PROGRAM Master1_IO_Map
VAR
	BYTE_AS_BIT_0: BYTE_AS_BIT;
	BYTE_AS_BIT_1: BYTE_AS_BIT;
	BYTE_AS_BIT_2: BYTE_AS_BIT;
	BYTE_AS_BIT_3: BYTE_AS_BIT;
	BYTE_AS_BIT_4: BYTE_AS_BIT;
	BYTE_AS_BIT_5: BYTE_AS_BIT;
	BYTE_AS_BIT_6: BYTE_AS_BIT;
	BYTE_AS_BIT_7: BYTE_AS_BIT;
	BYTE_AS_BIT_8: BYTE_AS_BIT;
	BYTE_AS_BIT_9: BYTE_AS_BIT;
	
	BIT_AS_BYTE_0: BIT_AS_BYTE;
	BIT_AS_BYTE_1: BIT_AS_BYTE;
	BIT_AS_BYTE_2: BIT_AS_BYTE;
	BIT_AS_BYTE_3: BIT_AS_BYTE;
	BIT_AS_BYTE_4: BIT_AS_BYTE;
	BIT_AS_BYTE_5: BIT_AS_BYTE;
	BIT_AS_BYTE_6: BIT_AS_BYTE;
	BIT_AS_BYTE_7: BIT_AS_BYTE;
	BIT_AS_BYTE_8: BIT_AS_BYTE;
	BIT_AS_BYTE_9: BIT_AS_BYTE;
	BIT_AS_BYTE_10: BIT_AS_BYTE;
	BIT_AS_BYTE_11: BIT_AS_BYTE;	
	
	OP10_MAS1_PORT1_BYTE1_DI_MODULE_1 AT %I* : BYTE;
	OP10_MAS1_PORT1_BYTE2_DI_MODULE_1 AT %I* : BYTE;
	OP10_MAS1_PORT2_BYTE1_DI_MODULE_2 AT %I* : BYTE;
	OP10_MAS1_PORT2_BYTE2_DI_MODULE_2 AT %I* : BYTE;
	OP10_MAS1_PORT3_BYTE1_DI_MODULE_3 AT %I* : BYTE;
	OP10_MAS1_PORT3_BYTE2_DI_MODULE_3 AT %I* : BYTE;
	OP10_MAS1_PORT4_BYTE1_DI_MODULE_4 AT %I* : BYTE;
	OP10_MAS1_PORT4_BYTE2_DI_MODULE_4 AT %I* : BYTE;
	OP10_MAS1_PORT5_BYTE1_DI_MODULE_5 AT %I* : BYTE;
	OP10_MAS1_PORT5_BYTE2_DI_MODULE_5 AT %I* : BYTE;
	
	OP10_MAS1_PORT6_BYTE1_DO_MODULE_1 AT %Q* : BYTE;
	OP10_MAS1_PORT6_BYTE2_DO_MODULE_1 AT %Q* : BYTE;
    OP10_MAS1_PORT6_BYTE3_DO_MODULE_1 AT %Q* : BYTE;
	OP10_MAS1_PORT6_BYTE4_DO_MODULE_1 AT %Q* : BYTE;
	
	OP10_MAS1_PORT7_BYTE1_DO_MODULE_2 AT %Q* : BYTE;
	OP10_MAS1_PORT7_BYTE2_DO_MODULE_2 AT %Q* : BYTE;
	OP10_MAS1_PORT7_BYTE3_DO_MODULE_2 AT %Q* : BYTE;
	OP10_MAS1_PORT7_BYTE4_DO_MODULE_2 AT %Q* : BYTE;
	
	OP10_MAS1_PORT8_BYTE1_DO_MODULE_3 AT %Q* : BYTE;
	OP10_MAS1_PORT8_BYTE2_DO_MODULE_3 AT %Q* : BYTE;
    OP10_MAS1_PORT8_BYTE3_DO_MODULE_3 AT %Q* : BYTE;
	OP10_MAS1_PORT8_BYTE4_DO_MODULE_3 AT %Q* : BYTE;
	
END_VAR

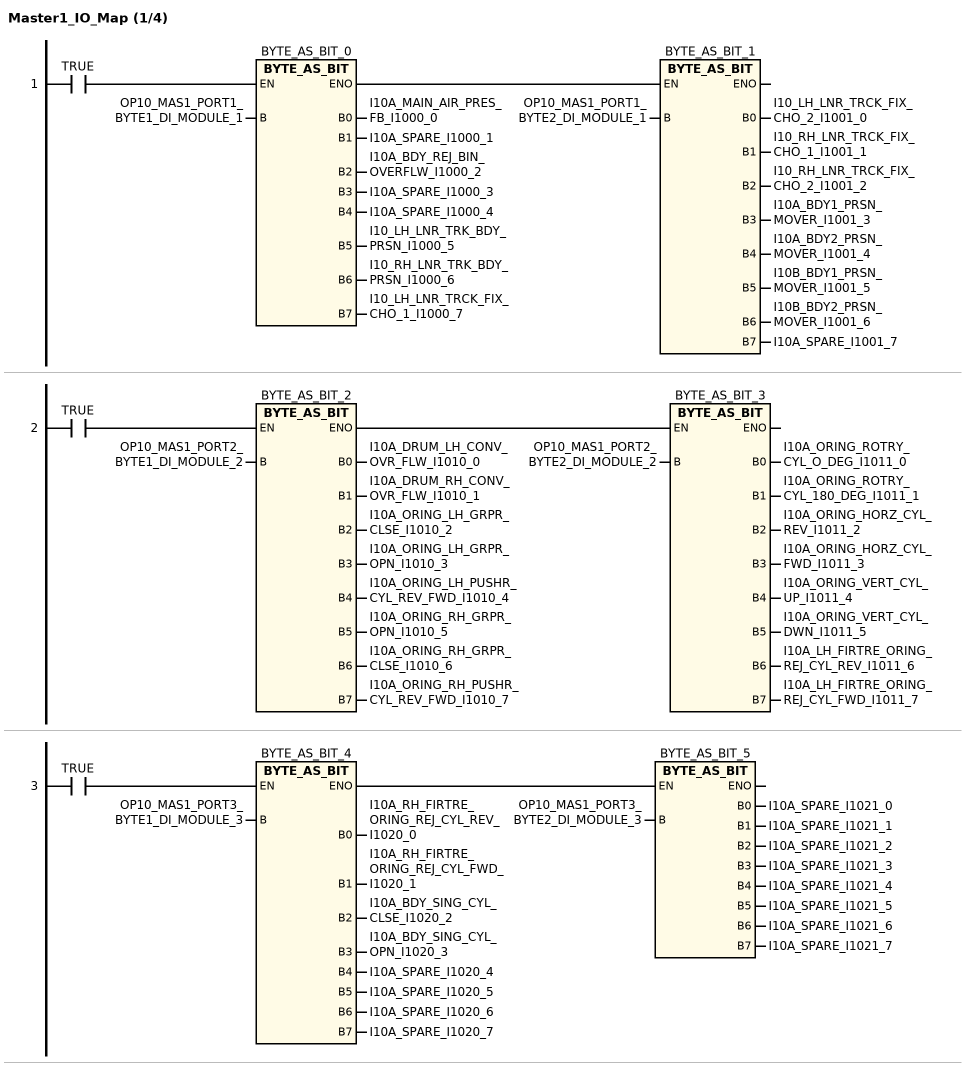
// NETWORK 1
BYTE_AS_BIT_0(
    B := OP10_MAS1_PORT1_BYTE1_DI_MODULE_1,
    B0 => I10A_MAIN_AIR_PRES_FB_I1000_0,
    B1 => I10A_SPARE_I1000_1,
    B2 => I10A_BDY_REJ_BIN_OVERFLW_I1000_2,
    B3 => I10A_SPARE_I1000_3,
    B4 => I10A_SPARE_I1000_4,
    B5 => I10_LH_LNR_TRK_BDY_PRSN_I1000_5,
    B6 => I10_RH_LNR_TRK_BDY_PRSN_I1000_6,
    B7 => I10_LH_LNR_TRCK_FIX_CHO_1_I1000_7); // BYTE_AS_BIT
BYTE_AS_BIT_1(
    B := OP10_MAS1_PORT1_BYTE2_DI_MODULE_1,
    B0 => I10_LH_LNR_TRCK_FIX_CHO_2_I1001_0,
    B1 => I10_RH_LNR_TRCK_FIX_CHO_1_I1001_1,
    B2 => I10_RH_LNR_TRCK_FIX_CHO_2_I1001_2,
    B3 => I10A_BDY1_PRSN_MOVER_I1001_3,
    B4 => I10A_BDY2_PRSN_MOVER_I1001_4,
    B5 => I10B_BDY1_PRSN_MOVER_I1001_5,
    B6 => I10B_BDY2_PRSN_MOVER_I1001_6,
    B7 => I10A_SPARE_I1001_7); // BYTE_AS_BIT

// NETWORK 2
BYTE_AS_BIT_2(
    B := OP10_MAS1_PORT2_BYTE1_DI_MODULE_2,
    B0 => I10A_DRUM_LH_CONV_OVR_FLW_I1010_0,
    B1 => I10A_DRUM_RH_CONV_OVR_FLW_I1010_1,
    B2 => I10A_ORING_LH_GRPR_CLSE_I1010_2,
    B3 => I10A_ORING_LH_GRPR_OPN_I1010_3,
    B4 => I10A_ORING_LH_PUSHR_CYL_REV_FWD_I1010_4,
    B5 => I10A_ORING_RH_GRPR_OPN_I1010_5,
    B6 => I10A_ORING_RH_GRPR_CLSE_I1010_6,
    B7 => I10A_ORING_RH_PUSHR_CYL_REV_FWD_I1010_7); // BYTE_AS_BIT
BYTE_AS_BIT_3(
    B := OP10_MAS1_PORT2_BYTE2_DI_MODULE_2,
    B0 => I10A_ORING_ROTRY_CYL_O_DEG_I1011_0,
    B1 => I10A_ORING_ROTRY_CYL_180_DEG_I1011_1,
    B2 => I10A_ORING_HORZ_CYL_REV_I1011_2,
    B3 => I10A_ORING_HORZ_CYL_FWD_I1011_3,
    B4 => I10A_ORING_VERT_CYL_UP_I1011_4,
    B5 => I10A_ORING_VERT_CYL_DWN_I1011_5,
    B6 => I10A_LH_FIRTRE_ORING_REJ_CYL_REV_I1011_6,
    B7 => I10A_LH_FIRTRE_ORING_REJ_CYL_FWD_I1011_7); // BYTE_AS_BIT

// NETWORK 3
BYTE_AS_BIT_4(
    B := OP10_MAS1_PORT3_BYTE1_DI_MODULE_3,
    B0 => I10A_RH_FIRTRE_ORING_REJ_CYL_REV_I1020_0,
    B1 => I10A_RH_FIRTRE_ORING_REJ_CYL_FWD_I1020_1,
    B2 => I10A_BDY_SING_CYL_CLSE_I1020_2,
    B3 => I10A_BDY_SING_CYL_OPN_I1020_3,
    B4 => I10A_SPARE_I1020_4,
    B5 => I10A_SPARE_I1020_5,
    B6 => I10A_SPARE_I1020_6,
    B7 => I10A_SPARE_I1020_7); // BYTE_AS_BIT
BYTE_AS_BIT_5(
    B := OP10_MAS1_PORT3_BYTE2_DI_MODULE_3,
    B0 => I10A_SPARE_I1021_0,
    B1 => I10A_SPARE_I1021_1,
    B2 => I10A_SPARE_I1021_2,
    B3 => I10A_SPARE_I1021_3,
    B4 => I10A_SPARE_I1021_4,
    B5 => I10A_SPARE_I1021_5,
    B6 => I10A_SPARE_I1021_6,
    B7 => I10A_SPARE_I1021_7); // BYTE_AS_BIT

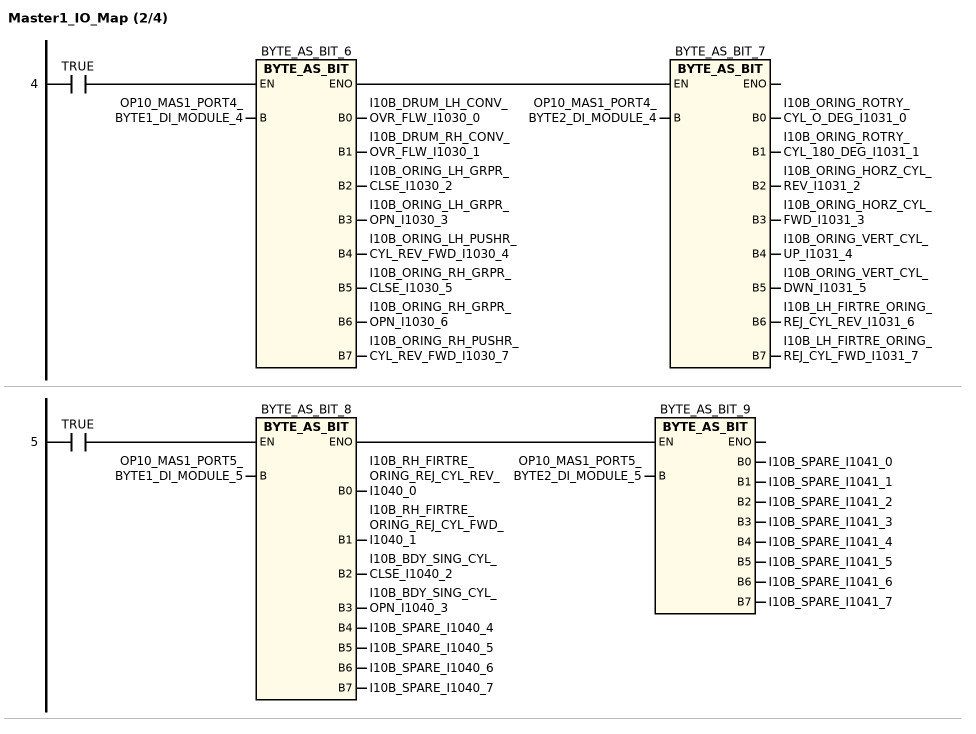
// NETWORK 4
BYTE_AS_BIT_6(
    B := OP10_MAS1_PORT4_BYTE1_DI_MODULE_4,
    B0 => I10B_DRUM_LH_CONV_OVR_FLW_I1030_0,
    B1 => I10B_DRUM_RH_CONV_OVR_FLW_I1030_1,
    B2 => I10B_ORING_LH_GRPR_CLSE_I1030_2,
    B3 => I10B_ORING_LH_GRPR_OPN_I1030_3,
    B4 => I10B_ORING_LH_PUSHR_CYL_REV_FWD_I1030_4,
    B5 => I10B_ORING_RH_GRPR_CLSE_I1030_5,
    B6 => I10B_ORING_RH_GRPR_OPN_I1030_6,
    B7 => I10B_ORING_RH_PUSHR_CYL_REV_FWD_I1030_7); // BYTE_AS_BIT
BYTE_AS_BIT_7(
    B := OP10_MAS1_PORT4_BYTE2_DI_MODULE_4,
    B0 => I10B_ORING_ROTRY_CYL_O_DEG_I1031_0,
    B1 => I10B_ORING_ROTRY_CYL_180_DEG_I1031_1,
    B2 => I10B_ORING_HORZ_CYL_REV_I1031_2,
    B3 => I10B_ORING_HORZ_CYL_FWD_I1031_3,
    B4 => I10B_ORING_VERT_CYL_UP_I1031_4,
    B5 => I10B_ORING_VERT_CYL_DWN_I1031_5,
    B6 => I10B_LH_FIRTRE_ORING_REJ_CYL_REV_I1031_6,
    B7 => I10B_LH_FIRTRE_ORING_REJ_CYL_FWD_I1031_7); // BYTE_AS_BIT

// NETWORK 5
BYTE_AS_BIT_8(
    B := OP10_MAS1_PORT5_BYTE1_DI_MODULE_5,
    B0 => I10B_RH_FIRTRE_ORING_REJ_CYL_REV_I1040_0,
    B1 => I10B_RH_FIRTRE_ORING_REJ_CYL_FWD_I1040_1,
    B2 => I10B_BDY_SING_CYL_CLSE_I1040_2,
    B3 => I10B_BDY_SING_CYL_OPN_I1040_3,
    B4 => I10B_SPARE_I1040_4,
    B5 => I10B_SPARE_I1040_5,
    B6 => I10B_SPARE_I1040_6,
    B7 => I10B_SPARE_I1040_7); // BYTE_AS_BIT
BYTE_AS_BIT_9(
    B := OP10_MAS1_PORT5_BYTE2_DI_MODULE_5,
    B0 => I10B_SPARE_I1041_0,
    B1 => I10B_SPARE_I1041_1,
    B2 => I10B_SPARE_I1041_2,
    B3 => I10B_SPARE_I1041_3,
    B4 => I10B_SPARE_I1041_4,
    B5 => I10B_SPARE_I1041_5,
    B6 => I10B_SPARE_I1041_6,
    B7 => I10B_SPARE_I1041_7); // BYTE_AS_BIT

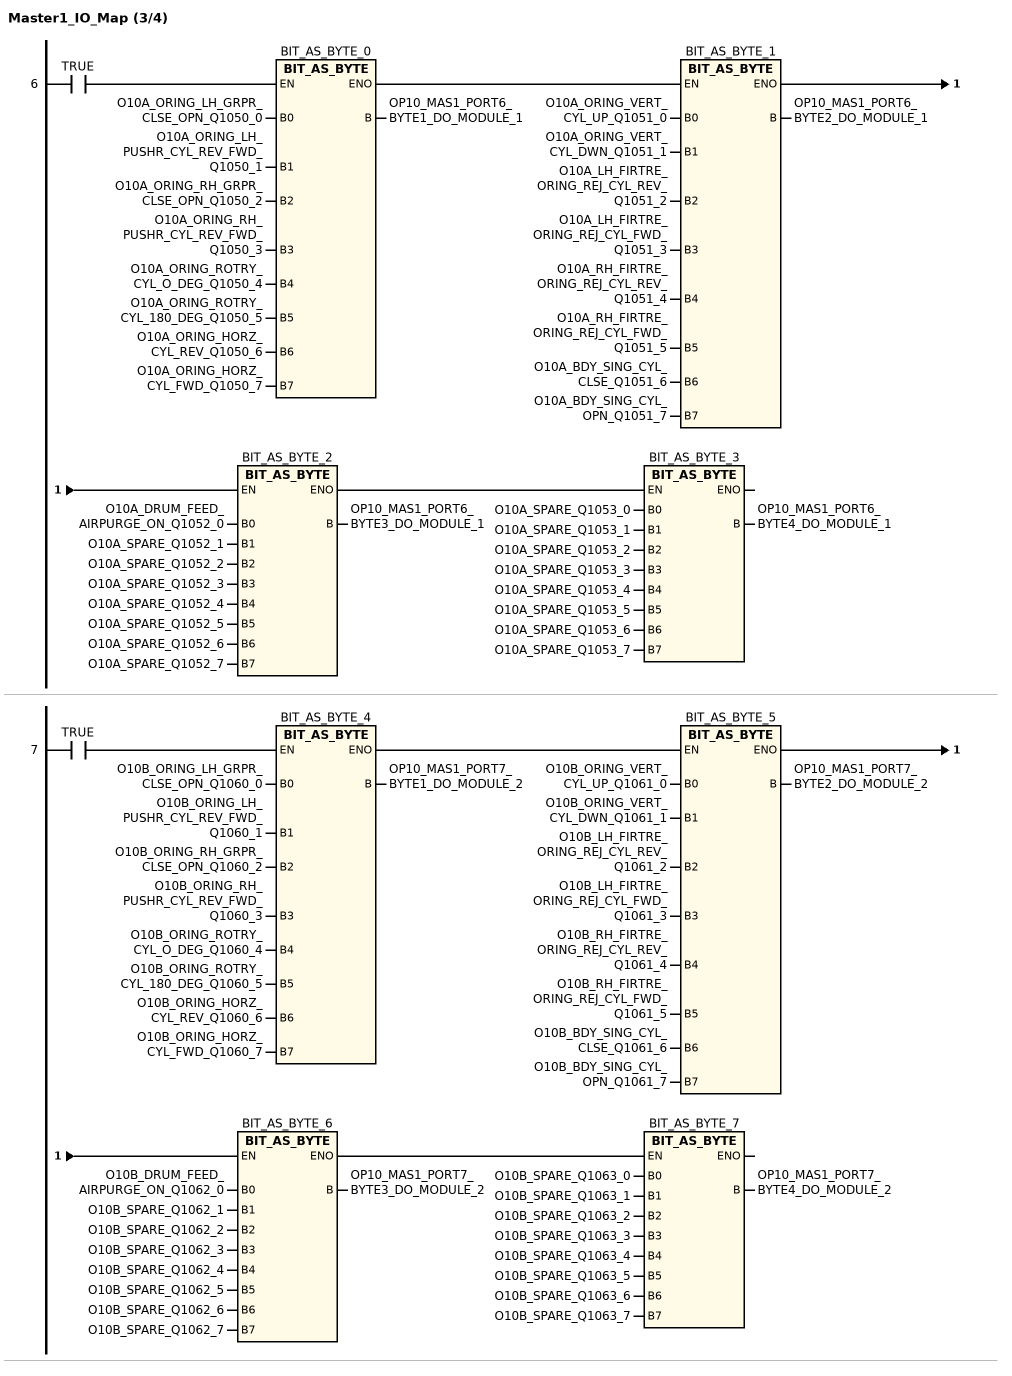
// NETWORK 6
BIT_AS_BYTE_0(
    B0 := O10A_ORING_LH_GRPR_CLSE_OPN_Q1050_0,
    B1 := O10A_ORING_LH_PUSHR_CYL_REV_FWD_Q1050_1,
    B2 := O10A_ORING_RH_GRPR_CLSE_OPN_Q1050_2,
    B3 := O10A_ORING_RH_PUSHR_CYL_REV_FWD_Q1050_3,
    B4 := O10A_ORING_ROTRY_CYL_O_DEG_Q1050_4,
    B5 := O10A_ORING_ROTRY_CYL_180_DEG_Q1050_5,
    B6 := O10A_ORING_HORZ_CYL_REV_Q1050_6,
    B7 := O10A_ORING_HORZ_CYL_FWD_Q1050_7,
    B => OP10_MAS1_PORT6_BYTE1_DO_MODULE_1); // BIT_AS_BYTE
BIT_AS_BYTE_1(
    B0 := O10A_ORING_VERT_CYL_UP_Q1051_0,
    B1 := O10A_ORING_VERT_CYL_DWN_Q1051_1,
    B2 := O10A_LH_FIRTRE_ORING_REJ_CYL_REV_Q1051_2,
    B3 := O10A_LH_FIRTRE_ORING_REJ_CYL_FWD_Q1051_3,
    B4 := O10A_RH_FIRTRE_ORING_REJ_CYL_REV_Q1051_4,
    B5 := O10A_RH_FIRTRE_ORING_REJ_CYL_FWD_Q1051_5,
    B6 := O10A_BDY_SING_CYL_CLSE_Q1051_6,
    B7 := O10A_BDY_SING_CYL_OPN_Q1051_7,
    B => OP10_MAS1_PORT6_BYTE2_DO_MODULE_1); // BIT_AS_BYTE
BIT_AS_BYTE_2(
    B0 := O10A_DRUM_FEED_AIRPURGE_ON_Q1052_0,
    B1 := O10A_SPARE_Q1052_1,
    B2 := O10A_SPARE_Q1052_2,
    B3 := O10A_SPARE_Q1052_3,
    B4 := O10A_SPARE_Q1052_4,
    B5 := O10A_SPARE_Q1052_5,
    B6 := O10A_SPARE_Q1052_6,
    B7 := O10A_SPARE_Q1052_7,
    B => OP10_MAS1_PORT6_BYTE3_DO_MODULE_1); // BIT_AS_BYTE
BIT_AS_BYTE_3(
    B0 := O10A_SPARE_Q1053_0,
    B1 := O10A_SPARE_Q1053_1,
    B2 := O10A_SPARE_Q1053_2,
    B3 := O10A_SPARE_Q1053_3,
    B4 := O10A_SPARE_Q1053_4,
    B5 := O10A_SPARE_Q1053_5,
    B6 := O10A_SPARE_Q1053_6,
    B7 := O10A_SPARE_Q1053_7,
    B => OP10_MAS1_PORT6_BYTE4_DO_MODULE_1); // BIT_AS_BYTE

// NETWORK 7
BIT_AS_BYTE_4(
    B0 := O10B_ORING_LH_GRPR_CLSE_OPN_Q1060_0,
    B1 := O10B_ORING_LH_PUSHR_CYL_REV_FWD_Q1060_1,
    B2 := O10B_ORING_RH_GRPR_CLSE_OPN_Q1060_2,
    B3 := O10B_ORING_RH_PUSHR_CYL_REV_FWD_Q1060_3,
    B4 := O10B_ORING_ROTRY_CYL_O_DEG_Q1060_4,
    B5 := O10B_ORING_ROTRY_CYL_180_DEG_Q1060_5,
    B6 := O10B_ORING_HORZ_CYL_REV_Q1060_6,
    B7 := O10B_ORING_HORZ_CYL_FWD_Q1060_7,
    B => OP10_MAS1_PORT7_BYTE1_DO_MODULE_2); // BIT_AS_BYTE
BIT_AS_BYTE_5(
    B0 := O10B_ORING_VERT_CYL_UP_Q1061_0,
    B1 := O10B_ORING_VERT_CYL_DWN_Q1061_1,
    B2 := O10B_LH_FIRTRE_ORING_REJ_CYL_REV_Q1061_2,
    B3 := O10B_LH_FIRTRE_ORING_REJ_CYL_FWD_Q1061_3,
    B4 := O10B_RH_FIRTRE_ORING_REJ_CYL_REV_Q1061_4,
    B5 := O10B_RH_FIRTRE_ORING_REJ_CYL_FWD_Q1061_5,
    B6 := O10B_BDY_SING_CYL_CLSE_Q1061_6,
    B7 := O10B_BDY_SING_CYL_OPN_Q1061_7,
    B => OP10_MAS1_PORT7_BYTE2_DO_MODULE_2); // BIT_AS_BYTE
BIT_AS_BYTE_6(
    B0 := O10B_DRUM_FEED_AIRPURGE_ON_Q1062_0,
    B1 := O10B_SPARE_Q1062_1,
    B2 := O10B_SPARE_Q1062_2,
    B3 := O10B_SPARE_Q1062_3,
    B4 := O10B_SPARE_Q1062_4,
    B5 := O10B_SPARE_Q1062_5,
    B6 := O10B_SPARE_Q1062_6,
    B7 := O10B_SPARE_Q1062_7,
    B => OP10_MAS1_PORT7_BYTE3_DO_MODULE_2); // BIT_AS_BYTE
BIT_AS_BYTE_7(
    B0 := O10B_SPARE_Q1063_0,
    B1 := O10B_SPARE_Q1063_1,
    B2 := O10B_SPARE_Q1063_2,
    B3 := O10B_SPARE_Q1063_3,
    B4 := O10B_SPARE_Q1063_4,
    B5 := O10B_SPARE_Q1063_5,
    B6 := O10B_SPARE_Q1063_6,
    B7 := O10B_SPARE_Q1063_7,
    B => OP10_MAS1_PORT7_BYTE4_DO_MODULE_2); // BIT_AS_BYTE

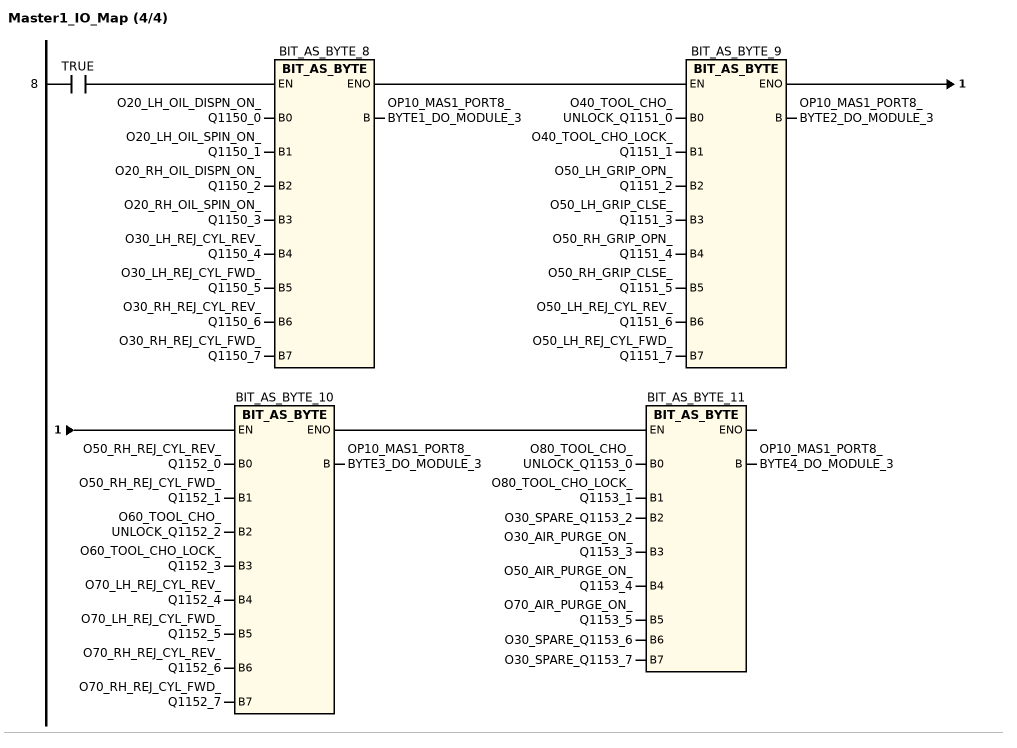
// NETWORK 8
BIT_AS_BYTE_8(
    B0 := O20_LH_OIL_DISPN_ON_Q1150_0,
    B1 := O20_LH_OIL_SPIN_ON_Q1150_1,
    B2 := O20_RH_OIL_DISPN_ON_Q1150_2,
    B3 := O20_RH_OIL_SPIN_ON_Q1150_3,
    B4 := O30_LH_REJ_CYL_REV_Q1150_4,
    B5 := O30_LH_REJ_CYL_FWD_Q1150_5,
    B6 := O30_RH_REJ_CYL_REV_Q1150_6,
    B7 := O30_RH_REJ_CYL_FWD_Q1150_7,
    B => OP10_MAS1_PORT8_BYTE1_DO_MODULE_3); // BIT_AS_BYTE
BIT_AS_BYTE_9(
    B0 := O40_TOOL_CHO_UNLOCK_Q1151_0,
    B1 := O40_TOOL_CHO_LOCK_Q1151_1,
    B2 := O50_LH_GRIP_OPN_Q1151_2,
    B3 := O50_LH_GRIP_CLSE_Q1151_3,
    B4 := O50_RH_GRIP_OPN_Q1151_4,
    B5 := O50_RH_GRIP_CLSE_Q1151_5,
    B6 := O50_LH_REJ_CYL_REV_Q1151_6,
    B7 := O50_LH_REJ_CYL_FWD_Q1151_7,
    B => OP10_MAS1_PORT8_BYTE2_DO_MODULE_3); // BIT_AS_BYTE
BIT_AS_BYTE_10(
    B0 := O50_RH_REJ_CYL_REV_Q1152_0,
    B1 := O50_RH_REJ_CYL_FWD_Q1152_1,
    B2 := O60_TOOL_CHO_UNLOCK_Q1152_2,
    B3 := O60_TOOL_CHO_LOCK_Q1152_3,
    B4 := O70_LH_REJ_CYL_REV_Q1152_4,
    B5 := O70_LH_REJ_CYL_FWD_Q1152_5,
    B6 := O70_RH_REJ_CYL_REV_Q1152_6,
    B7 := O70_RH_REJ_CYL_FWD_Q1152_7,
    B => OP10_MAS1_PORT8_BYTE3_DO_MODULE_3); // BIT_AS_BYTE
BIT_AS_BYTE_11(
    B0 := O80_TOOL_CHO_UNLOCK_Q1153_0,
    B1 := O80_TOOL_CHO_LOCK_Q1153_1,
    B2 := O30_SPARE_Q1153_2,
    B3 := O30_AIR_PURGE_ON_Q1153_3,
    B4 := O50_AIR_PURGE_ON_Q1153_4,
    B5 := O70_AIR_PURGE_ON_Q1153_5,
    B6 := O30_SPARE_Q1153_6,
    B7 := O30_SPARE_Q1153_7,
    B => OP10_MAS1_PORT8_BYTE4_DO_MODULE_3); // BIT_AS_BYTE

END_PROGRAM

(* stored: Version 1.1.0.1, ProductVersion 3.1.4024.11
   POU Master1_IO_Map: Id {263a00eb-fffc-4145-a524-ff0099822003}, SpecialFunc None *)
